FUNCTION_BLOCK FB_LamparaMemorizada_LD_2
// La lampara se enciende al accionar el pulsador de conexion
// La lampara se apaga al accionar el pulsador de desconexion
VAR
    Memoria: RS;
    Lampara AT %Q*: BOOL;
    PulsadorConexion AT %I*: BOOL;
    PulsadorDesconexion AT %I*: BOOL;
END_VAR

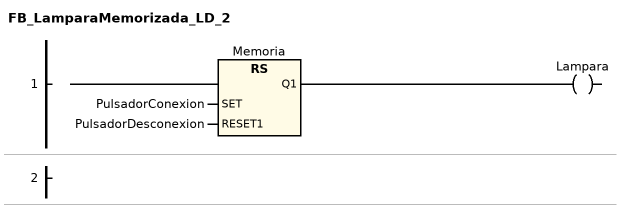
// NETWORK 1
Memoria(SET := PulsadorConexion, RESET1 := PulsadorDesconexion); // RS
Lampara := Memoria.Q1;

// NETWORK 2

END_FUNCTION_BLOCK

(* stored: Version 1.1.0.1, ProductVersion 3.1.4024.15
   POU FB_LamparaMemorizada_LD_2: Id {a023541f-9843-42f8-af59-58d4e714d522}, SpecialFunc None *)
